// TwinCAT 3 PLC project Untitled1
// ProgramVersion: 3.1.4023.0
// libraries:
//   Tc2_MC2, * (Beckhoff Automation GmbH)
//   Tc2_NC, * (Beckhoff Automation GmbH)
//   Tc2_NCI, * (Beckhoff Automation GmbH)
//   Tc2_PlcInterpolation, * (Beckhoff Automation GmbH)
//   Tc2_Standard, * (Beckhoff Automation GmbH)
//   Tc2_System, * (Beckhoff Automation GmbH)
//   Tc3_Module, * (Beckhoff Automation GmbH)
//   Tc3_mxAutomation, * (Beckhoff Automation GmbH)
//   Tc3_mxAutomationV3_0, * (Beckhoff Automation GmbH)
//   Tc3_mxAutomationV3_1, * (Beckhoff Automation GmbH)
//   Tc3_mxAutomationV3_2, * (Beckhoff Automation GmbH)
//   Tc3_uniValPlc, * (Beckhoff Automation GmbH)
//   Tc3_uniValPlc_v4, * (Beckhoff Automation GmbH)
//   Tc3_uniValPlc_v4_3, * (Beckhoff Automation GmbH)
//   Tc3_uniValPlc_v4_4, * (Beckhoff Automation GmbH)
//   Tc3_uniValPlc_v4_5, * (Beckhoff Automation GmbH)
// project tree:
//   DUTs/ AxisFeedback.TcDUT, AxisInputs.TcDUT
//   GVLs/ Feedback.TcGVL, Inputs.TcGVL, NCI.TcGVL
//   / PlcTask.TcTTO
//   POUs/ AxisControl.TcPOU, FB_EnableAxes.TcPOU, FB_NciFastMFunctions.TcPOU, FB_NciMFunctions.TcPOU, FB_SimpleNciSequence.TcPOU, MAIN.TcPOU, PRG_MFuncControl.TcPOU
// real-time tasks:
//   TASK PlcTask: cycle T#10ms, priority 20, ADS port 350
// motion (NC):
//   TASK NC-Task 1 SAF: cycle T#2ms, priority 4, ADS port 501
//   TASK NC-Task 1 SVB: cycle T#10ms, priority 8, ADS port 511
//   AXIS X (id 1)
//     Dynamic: Acceleration=1505, Deceleration=1505
//     OtherSettings: AllowMotionCmdToSlave=true
//     encoder EncType=1
//     drive DrvType=5
//       TimeComp: TaskDelayCycles=1
//     controller CtrType=1
//       CtrPara: PriorControlFactor=1
//         Observer: BandWidth=20
//   AXIS Y (id 2)
//     OtherSettings: AllowMotionCmdToSlave=true
//     encoder EncType=1
//     drive DrvType=5
//       TimeComp: TaskDelayCycles=1
//     controller CtrType=1
//       CtrPara: PriorControlFactor=1
//         Observer: BandWidth=20
//   AXIS Z (id 3)
//     OtherSettings: AllowMotionCmdToSlave=true
//     encoder EncType=1
//     drive DrvType=5
//       TimeComp: TaskDelayCycles=1
//     controller CtrType=1
//       CtrPara: PriorControlFactor=1
//         Observer: BandWidth=20
//   AXIS Q1 (id 4)
//     Dynamic: VeloJumpFactor=20, ToleranceBallAuxAxis=5
//     OtherSettings: AllowMotionCmdToSlave=true
//     encoder EncType=1
//     drive DrvType=5
//       TimeComp: TaskDelayCycles=1
//     controller CtrType=1
//       CtrPara: PriorControlFactor=1
//         Observer: BandWidth=20
//   AXIS Q2 (id 5)
//     OtherSettings: AllowMotionCmdToSlave=true
//     encoder EncType=1
//     drive DrvType=5
//       TimeComp: TaskDelayCycles=1
//     controller CtrType=1
//       CtrPara: PriorControlFactor=1
//         Observer: BandWidth=20
//   AXIS Q3 (id 6)
//     OtherSettings: AllowMotionCmdToSlave=true
//     encoder EncType=1
//     drive DrvType=5
//       TimeComp: TaskDelayCycles=1
//     controller CtrType=1
//       CtrPara: PriorControlFactor=1
//         Observer: BandWidth=20
// variable links:
//   Untitled1/Untitled1 Instance <-> NC-Task 1 SAF/Axes/Q1
//     PlcTask Inputs/MAIN.io_Q1.NcToPlc <-> Outputs/ToPlc
//     PlcTask Outputs/MAIN.io_Q1.PlcToNc <-> Inputs/FromPlc
//   Untitled1/Untitled1 Instance <-> NC-Task 1 SAF/Axes/Q2
//     PlcTask Inputs/MAIN.io_Q2.NcToPlc <-> Outputs/ToPlc
//     PlcTask Outputs/MAIN.io_Q2.PlcToNc <-> Inputs/FromPlc
//   Untitled1/Untitled1 Instance <-> NC-Task 1 SAF/Axes/Q3
//     PlcTask Inputs/MAIN.io_Q3.NcToPlc <-> Outputs/ToPlc
//     PlcTask Outputs/MAIN.io_Q3.PlcToNc <-> Inputs/FromPlc
//   Untitled1/Untitled1 Instance <-> NC-Task 1 SAF/Axes/X
//     PlcTask Inputs/MAIN.io_X.NcToPlc <-> Outputs/ToPlc
//     PlcTask Outputs/MAIN.io_X.PlcToNc <-> Inputs/FromPlc
//   Untitled1/Untitled1 Instance <-> NC-Task 1 SAF/Axes/Y
//     PlcTask Inputs/MAIN.io_Y.NcToPlc <-> Outputs/ToPlc
//     PlcTask Outputs/MAIN.io_Y.PlcToNc <-> Inputs/FromPlc
//   Untitled1/Untitled1 Instance <-> NC-Task 1 SAF/Axes/Z
//     PlcTask Inputs/MAIN.io_Z.NcToPlc <-> Outputs/ToPlc
//     PlcTask Outputs/MAIN.io_Z.PlcToNc <-> Inputs/FromPlc
//   Untitled1/Untitled1 Instance <-> NC-Task 1 SAF/Interpolation
//     PlcTask Inputs/MAIN.in_stItpToPlc <-> Outputs/ToPlc
//     PlcTask Outputs/MAIN.out_stPlcToItp <-> Inputs/FromPlc

CONFIGURATION Untitled1
    RESOURCE PLC ON TwinCAT3
        TASK PlcTask(INTERVAL := T#10ms, PRIORITY := 20);
        PROGRAM MAIN WITH PlcTask : MAIN;
    END_RESOURCE
END_CONFIGURATION

// ---- DUTs/AxisFeedback.TcDUT
TYPE AxisFeedback :
STRUCT
	Status			: BOOL;
	Busy			: BOOL;
	Active			: BOOL;
	Error			: BOOL;
	ErrorID			: UDINT;	
	Done			: BOOL;
	CommandAborted	: BOOL;
END_STRUCT
END_TYPE

// ---- DUTs/AxisInputs.TcDUT
TYPE AxisInputs :
STRUCT
	PowerEnable		: BOOL;
	EnablePositive	: BOOL;
	EnableNegative  : BOOL;
	Override		: LREAL;
	BufferMode		: MC_BufferMode;
	Options			: ST_PowerOptions;
	
	ResetEnable		: BOOL;
	
	StopExecute			: BOOL;
	StopDeceleration	: LREAL;
	StopJerk			: LREAL;
	StopOptions			: ST_MoveOptions;
	
	
	JogForward		: BOOL;
	JogBackward		: BOOL;
	jogMode			: E_JogMode;
	JogPosition		: LREAL;
	JogVelocity		: LREAL;
	JogAcceleration : LREAL;
	JogDeceleration : LREAL;
	JogJerk			: LREAL;
	
	HaltExecute			: BOOL;
	HaltDeceleration	: LREAL;
	HaltJerk			: LREAL;
	HaltBufferMode		: MC_BufferMode;
	HaltOptions			: ST_MoveOptions;
	
	MoveAbsoluteExecute				: BOOL;
	MoveAbsolutePosition			: LREAL;
	MoveAbsoluteVelocity			: LREAL;
	MoveAbsoluteAcceleration		: LREAL;
	MoveAbsoluteDeceleration		: LREAL;
	MoveAbsoluteJerk				: LREAL;
	MoveAbsoluteBufferMode			: MC_BufferMode;
	MoveAbsoluteOptions				: ST_MoveOptions;
	
	MoveRelativeExecute				: BOOL;
	MoveRelativeDistance			: LREAL;
	MoveRelativeVelocity			: LREAL;
	MoveRelativeAcceleration		: LREAL;
	MoveRelativeDeceleration		: LREAL;
	MoveRelativeJerk				: LREAL;
	MoveRelativeBufferMode			: MC_BufferMode;
	MoveRelativeOptions				: ST_MoveOptions;

END_STRUCT
END_TYPE

// ---- GVLs/Feedback.TcGVL
{attribute 'qualified_only'}
VAR_GLOBAL
	AxisX_Feedback		: AxisFeedback;
	AxisY_Feedback		: AxisFeedback;
	AxisZ_Feedback		: AxisFeedback;
END_VAR

// ---- GVLs/Inputs.TcGVL
{attribute 'qualified_only'}
VAR_GLOBAL
	AxisX_Inputs		: AxisInputs;
	AxisY_Inputs		: AxisInputs;
	AxisZ_Inputs		: AxisInputs;
END_VAR

// ---- GVLs/NCI.TcGVL
{attribute 'qualified_only'}
VAR_GLOBAL
	bMFunc					: ARRAY[0..cnMaxMFuncNumber] OF BOOL;
	bQuitMFunc				: ARRAY[0..cnMaxMFuncNumber] OF BOOL;
	bFastMFunc				: ARRAY[0..cnMaxMFuncNumber] OF BOOL;
END_VAR
VAR_GLOBAL CONSTANT
	cnMaxMFuncNumber		: INT	:= 159;
END_VAR

// ---- POUs/MAIN.TcPOU
PROGRAM MAIN
VAR
	bUserEnableAxes			:	BOOL	:= TRUE;
	fUserOverride			:	LREAL	:= 100.0;
	
	io_X					:	AXIS_REF;
	io_Y					:	AXIS_REF;
	io_Z					:	AXIS_REF;
	io_Q1					:	AXIS_REF;
	io_Q2					:	AXIS_REF;
	io_Q3					:	AXIS_REF;
	
	in_stItpToPlc	AT %I*	:	NcToPlc_NciChannel_Ref;
	out_stPlcToItp	AT %Q*	:	PLCTONC_NCICHANNEL_REF;

	fbEnableAxes			:	FB_EnableAxes;
	bAllAxesReady			:	BOOL;
	
	
	fbSimpleNciSequence		:	FB_SimpleNciSequence;
	bExecSimpleNci			:	BOOL	:= FALSE;
END_VAR

fbEnableAxes(
	bEnableAxes	:= bUserEnableAxes, 
	stX			:=io_X , 
	stY			:=io_Y , 
	stZ			:=io_Z , 
	stM1		:=io_Q1 , 
	stM2		:=io_Q2 , 
	stM3		:=io_Q3 , 
	bAllAxesReady => bAllAxesReady );
	
ItpSetOverridePercent(fOverridePercent:=fUserOverride , sPlcToNci:=out_stPlcToItp);

fbSimpleNciSequence(
	bExecute	:= bExecSimpleNci, 
	bBusy		=> , 
	bError		=> , 
	bDone		=> , 
	stX			:= io_X, 
	stY			:= io_Y, 
	stZ			:= io_Z, 
	stQ1		:= io_Q1,
	stQ2		:= io_Q2,
	stQ3		:= io_Q3,
	stItpToPlc	:= in_stItpToPlc , 
	stPlcToItp	:= out_stPlcToItp);

END_PROGRAM

// ---- POUs/FB_EnableAxes.TcPOU
FUNCTION_BLOCK FB_EnableAxes
VAR_INPUT
	bEnableAxes: BOOL:= TRUE;
END_VAR
VAR_OUTPUT
	bAllAxesReady:	BOOL:= FALSE;
END_VAR
VAR_IN_OUT
	stX:	AXIS_REF;
	stY:	AXIS_REF;
	stZ:	AXIS_REF;
	stM1:	AXIS_REF;
	stM2:	AXIS_REF;
	stM3:	AXIS_REF;
END_VAR
VAR
	fOverride:	LREAL	:= 100.0;
	fbPowerX:	MC_Power;
	fbPowerY:	MC_Power;
	fbPowerZ:	MC_Power;
	fbPowerM1:	MC_Power;
	fbPowerM2:	MC_Power;
	fbPowerM3:	MC_Power;
END_VAR

stX.ReadStatus();
stY.ReadStatus();
stZ.ReadStatus();
stM1.ReadStatus();
stM2.ReadStatus();
stM3.ReadStatus();


fbPowerX(
	Enable:=bEnableAxes, 
	Enable_Positive:=bEnableAxes, 
	Enable_Negative:=bEnableAxes, 
	Override:=fOverride, 
	BufferMode:= , 
	Axis:=stX, 
	Status=> , 
	Busy=> , 
	Active=> , 
	Error=> , 
	ErrorID=> );
fbPowerY(
	Enable:=bEnableAxes, 
	Enable_Positive:=bEnableAxes, 
	Enable_Negative:=bEnableAxes, 
	Override:=fOverride, 
	BufferMode:= , 
	Axis:=stY, 
	Status=> , 
	Busy=> , 
	Active=> , 
	Error=> , 
	ErrorID=> );	
fbPowerZ(
	Enable:=bEnableAxes, 
	Enable_Positive:=bEnableAxes, 
	Enable_Negative:=bEnableAxes, 
	Override:=fOverride, 
	BufferMode:= , 
	Axis:=stZ, 
	Status=> , 
	Busy=> , 
	Active=> , 
	Error=> , 
	ErrorID=> );	
fbPowerM1(
	Enable:=bEnableAxes, 
	Enable_Positive:=bEnableAxes, 
	Enable_Negative:=bEnableAxes, 
	Override:=fOverride, 
	BufferMode:= , 
	Axis:=stM1, 
	Status=> , 
	Busy=> , 
	Active=> , 
	Error=> , 
	ErrorID=> );	
fbPowerM2(
	Enable:=bEnableAxes, 
	Enable_Positive:=bEnableAxes, 
	Enable_Negative:=bEnableAxes, 
	Override:=fOverride, 
	BufferMode:= , 
	Axis:=stM2, 
	Status=> , 
	Busy=> , 
	Active=> , 
	Error=> , 
	ErrorID=> );	
fbPowerM3(
	Enable:=bEnableAxes, 
	Enable_Positive:=bEnableAxes, 
	Enable_Negative:=bEnableAxes, 
	Override:=fOverride, 
	BufferMode:= , 
	Axis:=stM3, 
	Status=> , 
	Busy=> , 
	Active=> , 
	Error=> , 
	ErrorID=> );	
bAllAxesReady	:= fbPowerX.Status AND fbPowerY.Status AND fbPowerZ.Status AND 
	fbPowerM1.Status AND fbPowerM2.Status AND fbPowerM3.Status;

END_FUNCTION_BLOCK

// ---- POUs/FB_SimpleNciSequence.TcPOU
FUNCTION_BLOCK FB_SimpleNciSequence
VAR_INPUT
	bExecute			: BOOL;
END_VAR
VAR_OUTPUT
	bBusy				: BOOL;
	bError				: BOOL;
	bDone				: BOOL;
END_VAR
VAR_IN_OUT
	stX					: AXIS_REF;
	stY					: AXIS_REF;
	stZ					: AXIS_REF;
	stQ1				: AXIS_REF;
	stQ2				: AXIS_REF;
	stQ3				: AXIS_REF;
	stItpToPlc			: NCTOPLC_NCICHANNEL_REF;
	stPlcToItp			: PLCTONC_NCICHANNEL_REF;
END_VAR
VAR
	nState				: UDINT	:= 0;
	nErrorState			: UDINT;
	
	fbBuildGroup		: CfgBuildExt3DGroup;
	fbLoadGCode			: ItpLoadProgEx;
	fbStartGCode		: ItpStartStopEx;
	fbClearGroup		: CfgReconfigGroup;
	fbConfirmHsk		: ItpConfirmHsk;
	
	nInterpreterState	: UDINT	:= 0;
	bConfirmHsk			: BOOL	:= FALSE;
	
//	sPrgName			: STRING(255) := 'GST_SampleFunctions.nc'; //'first.nc';
	sPrgName			: STRING(255) := 'first.nc'; //'';
//	sPrgName			: STRING(255) := 'sample.nc'; //'';
//	sPrgName			: STRING(255) := 'functionsExample.nc'; //'';
	
	
END_VAR

CASE nState OF
0:
	IF bExecute THEN
		bBusy	:= TRUE;
		bDone	:= FALSE;
		bError	:= FALSE;
		nErrorState	:= nState;
		nState	:= 10;
	END_IF	
	
10:
	// first build interpolation group 
	nInterpreterState	:= ItpGetStateInterpreter(sNciToPlc:=stItpToPlc);
	IF nInterpreterState = Tc2_NCI.NCI_INTERPRETER_IDLE THEN
		fbBuildGroup(
			bExecute	:= TRUE, 
			nGroupId	:= ItpGetGroupId(sNciToPlc:=stItpToPlc) , 
			nXAxisId	:= stX.NcToPlc.AxisId, 
			nYAxisId	:= stY.NcToPlc.AxisId, 
			nZAxisId	:= stZ.NcToPlc.AxisId, 
			nQ1AxisId	:= stQ1.NcToPlc.AxisId, 
			nQ2AxisId	:= stQ2.NcToPlc.AxisId, 
			nQ3AxisId	:= stQ3.NcToPlc.AxisId, 
			nQ4AxisId	:= 0, 
			nQ5AxisId	:= 0, 
			tTimeOut	:= , 
			bBusy		=> , 
			bErr		=> , 
			nErrId		=> );
			
		IF NOT fbBuildGroup.bBusy THEN
			IF NOT fbBuildGroup.bErr THEN
				nState	:= 20;
			ELSE
				(* add error handling *)
				nErrorState	:= nState;
				bBusy	:= FALSE;
				bError	:= TRUE;
				nState	:= 9999;
			END_IF
			fbBuildGroup(bExecute:=FALSE); 
		END_IF
	END_IF
	
20:
	// load g-code file 
	// pls. ensure that first.nc is available in TwinCAT\MC\NCI-folder 
	fbLoadGCode(
		sNciToPlc	:= stItpToPlc, 
		bExecute	:= TRUE, 
		sPrg		:= sPrgName, 
		nLength		:= INT_TO_UDINT(LEN(sPrgName)), 
		tTimeOut	:= , 
		bBusy		=> , 
		bErr		=> , 
		nErrId		=> );
		
	IF NOT fbLoadGCode.bBusy THEN
		IF NOT fbLoadGCode.bErr THEN
			nState	:= 30;
		ELSE
			(* add error handling *)
			nErrorState	:= nState;
			bBusy	:= FALSE;
			bError	:= TRUE;
			nState	:= 9999;				
		END_IF
		fbLoadGCode(sNciToPlc:=stItpToPlc, bExecute:=FALSE); 
	END_IF
	
30:
	// we have to check the status of the interpreter. It has to be in ready state, in case of loading the program successfully.
	nInterpreterState	:= ItpGetStateInterpreter(sNciToPlc:=stItpToPlc);
	IF nInterpreterState = Tc2_NCI.NCI_INTERPRETER_READY THEN
		nState	:= 40;
	ELSE
		(* add error handling *)
		nErrorState	:= nState;
		bBusy	:= FALSE;
		bError	:= TRUE;
		nState	:= 9999;				
	END_IF
	
40:
	// start g-code file
	fbStartGCode(
		bStart		:=TRUE, 
		bStop		:=FALSE, 
		tTimeOut	:= , 
		sNciToPlc	:= stItpToPlc, 
		bBusy		=> , 
		bErr		=> , 
		nErrId		=> );
		
	IF NOT fbStartGCode.bBusy THEN
		IF NOT fbStartGCode.bErr THEN
			nState	:= 50;
		ELSE	
			(* add error handling *)
			nErrorState	:= nState;
			bBusy	:= FALSE;
			bError	:= TRUE;
			nState	:= 9999;				
		END_IF
		fbStartGCode( bStart:=FALSE, sNciToPlc:= stItpToPlc ); 
	END_IF
	
50:
	// check state, again - we are at least not in ready state for several ticks
	// this is to ensure that we don't indicate program has finished, before we have started 
	nInterpreterState	:= ItpGetStateInterpreter(sNciToPlc:=stItpToPlc);
	IF nInterpreterState <> Tc2_NCI.NCI_INTERPRETER_READY THEN
		// nci is running
		nState	:= 60;
	END_IF

60:
	nInterpreterState	:= ItpGetStateInterpreter(sNciToPlc:=stItpToPlc);
	IF	nInterpreterState = Tc2_NCI.NCI_INTERPRETER_READY THEN
		// program has finished
		nState	:= 70;
	ELSIF nInterpreterState = Tc2_NCI.NCI_INTERPRETER_ABORTED THEN
		// a run-time error occured - this could be a lag error or something else... 
		// add error handling
		;
	END_IF	
	
70:
	// program has finished 
	// now clear interpolation group 
	fbClearGroup(
		bExecute	:= TRUE, 
		nGroupId	:= ItpGetGroupId(sNciToPlc:=stItpToPlc) , 
		tTimeOut	:= , 
		bBusy		=> , 
		bErr		=> , 
		nErrId		=> );
		
	IF NOT fbClearGroup.bBusy THEN
		IF NOT fbClearGroup.bErr THEN
			nState	:= 80;
		ELSE
			(* add error handling *)
			nErrorState	:= nState;
			bBusy	:= FALSE;
			bError	:= TRUE;
			nState	:= 9999;				
		END_IF
		fbClearGroup(bExecute:=FALSE); 
	END_IF
80:
	bDone	:= TRUE;
	bBusy	:= FALSE;
	IF NOT bExecute THEN
		nState	:= 0;
	END_IF
	
9999:
	// error state 
	IF NOT bExecute THEN
		nState	:= 0;
		bError	:= FALSE;
	END_IF
END_CASE

// handling of m-functions is done outside statemachine
// all m-functions are directly confiremd. In a real application we have of course to consider the m-function numbers to turn on/off certain functions in the machine.
IF ItpIsHskMFunc(stItpToPlc) AND NOT fbConfirmHsk.bBusy THEN
	bConfirmHsk	:= TRUE;
ELSE	
	bConfirmHsk	:= FALSE;
END_IF	

fbConfirmHsk(
	bExecute:=bConfirmHsk , 
	sNciToPlc:=stItpToPlc , 
	sPlcToNci:=stPlcToItp , 
	bBusy=> , 
	bErr=> , 
	nErrId=> );

END_FUNCTION_BLOCK

// ---- POUs/AxisControl.TcPOU
FUNCTION_BLOCK AxisControl
VAR_INPUT
	Axis 			: AXIS_REF;
	AxisInputs		: AxisInputs;
END_VAR
VAR_OUTPUT
	Status			: AxisFeedback;
END_VAR
VAR
	Power			: MC_Power;
	Reset			: MC_Reset;
	Stop			: MC_Stop;
	Jog				: MC_Jog;
	Halt			: MC_Halt;
	MoveAbsolute	: MC_MoveAbsolute;
	MoveRelative	: MC_MoveRelative;
END_VAR

Power(Axis := Axis,
	  Enable := AxisInputs.PowerEnable,
	  Enable_Positive := AxisInputs.EnablePositive,
	  Enable_Negative := AxisInputs.EnableNegative,
	  Override := AxisInputs.Override,
	  BufferMode := AxisInputs.BufferMode,
	  Options := AxisInputs.Options,
	  Status => Status.Status,
	  Busy => Status.Busy,
	  Active => Status.Active,
	  Error => Status.Error,
	  ErrorID => Status.ErrorID);

	 
Reset(Axis := Axis,
	  Execute := AxisInputs.ResetEnable,
	  Done => Status.Done,
      Busy => Status.Busy,
	  Error => Status.Busy,
	  ErrorID => Status.ErrorID);
	  
Stop(Axis := Axis,
	 Execute := AxisInputs.StopExecute,
	 Deceleration := AxisInputs.StopDeceleration,
	 Jerk := AxisInputs.StopJerk,
	 Options := AxisInputs.StopOptions,
	 Done => Status.Done,
	 Busy => Status.Busy,
	 Active => Status.Active,
	 CommandAborted => Status.CommandAborted,
	 Error => Status.Error,
	 ErrorID => Status.ErrorID); 

Halt(Axis := Axis,
	 Execute := AxisInputs.HaltExecute,
	 Deceleration := AxisInputs.HaltDeceleration,
	 Jerk := AxisInputs.HaltJerk,
	 BufferMode := AxisInputs.HaltBufferMode,
	 Options := AxisInputs.HaltOptions,
	 Done => Status.Done,
	 Busy => Status.Busy,
	 Active => Status.Active,
	 CommandAborted => Status.CommandAborted,
	 Error => Status.Error,
	 ErrorID => Status.ErrorID); 

Jog(Axis := Axis,
	JogForward := AxisInputs.JogForward,
	JogBackwards := AxisInputs.JogBackward,
	Mode := AxisInputs.jogMode,
	Position := AxisInputs.JogPosition,
	Velocity := AxisInputs.JogVelocity,
	Acceleration := AxisInputs.JogAcceleration,
	Deceleration := AxisInputs.JogDeceleration,
	jerk := AxisInputs.JogJerk,
	Done => Status.Done,
	Busy => Status.Busy,
	Active => Status.Active,
	CommandAborted => Status.CommandAborted,
	Error => Status.Error,
	ErrorID => Status.ErrorID);
	
MoveAbsolute(Axis := Axis,
			 Execute := AxisInputs.MoveAbsoluteExecute,
			 Position := AxisInputs.MoveAbsolutePosition,
			 Acceleration := AxisInputs.MoveAbsoluteAcceleration,
			 Deceleration := AxisInputs.MoveAbsoluteDeceleration,
			 Jerk := AxisInputs.MoveAbsoluteJerk,
			 Options := AxisInputs.MoveAbsoluteOptions,
			 BufferMode := AxisInputs.MoveAbsoluteBufferMode,
			 Done => Status.Done,
			 Busy => Status.Busy,
			 Active => Status.Active,
			 CommandAborted => Status.CommandAborted,
			 Error => Status.Error,
			 ErrorID => Status.ErrorID);
				 
MoveRelative(Axis := Axis,
			 Execute := AxisInputs.MoveRelativeExecute,
			 Distance := AxisInputs.MoveRelativeDistance,
			 Acceleration := AxisInputs.MoveRelativeAcceleration,
			 Deceleration := AxisInputs.MoveRelativeDeceleration,
			 Jerk := AxisInputs.MoveRelativeJerk,
			 Options := AxisInputs.MoveRelativeOptions,
			 BufferMode := AxisInputs.MoveRelativeBufferMode,
			 Done => Status.Done,
			 Busy => Status.Busy,
			 Active => Status.Active,
			 CommandAborted => Status.CommandAborted,
			 Error => Status.Error,
			 ErrorID => Status.ErrorID);

END_FUNCTION_BLOCK

// ---- POUs/FB_NciFastMFunctions.TcPOU
FUNCTION_BLOCK FB_NciFastMFunctions
VAR_IN_OUT
	sNciToPlc		: NCTOPLC_NCICHANNEL_REF;
END_VAR
VAR_OUTPUT
END_VAR
VAR
	i				: INT;
	l				: SINT;
	bBit			: BOOL;
	index			: UINT;
END_VAR


(* Fill the global defined M-functions array with 
	fast M-Functions from NCI Channel *)

FOR i:=0 TO 4 DO  (* check all 5 dwords *)
	FOR l := 0 TO 31 DO
		bBit := GETBIT32(sNciToPlc.FastMFuncMask[i+1], l);
      	index := INT_TO_UINT((i*32) + l);
		IF ( bBit ) THEN
			NCI.bFastMFunc[index] := TRUE;
		ELSE
			NCI.bFastMFunc[index] := FALSE;
		END_IF
	END_FOR
END_FOR

END_FUNCTION_BLOCK

// ---- POUs/FB_NciMFunctions.TcPOU
FUNCTION_BLOCK FB_NciMFunctions
VAR_IN_OUT
	sNciToPlc		: NCTOPLC_NCICHANNEL_REF;
	sPlcToNci		: PLCTONC_NCICHANNEL_REF;
END_VAR
VAR_OUTPUT
	bBusy			: BOOL;
	bError			: BOOL;
	nErrorId		: UDINT;
END_VAR
VAR
	fbConfirm		: ItpConfirmHsk;
	nAktMfunc		: INT :=  -1;
	bConfirm		: BOOL;
	i				: INT;
END_VAR


(* Check for m function and store information in bMFunc Array	*)
IF ItpIsHskMFunc(sNciToPlc:= sNciToPlc) THEN
	nAktMfunc 			:= ItpGetHskMFunc(sNciToPlc:= sNciToPlc);
	NCI.bMFunc[nAktMfunc]	:= TRUE;
ELSE
	nAktMfunc 	:= -1;
	bConfirm 	:= FALSE;
	FOR i := 0 TO NCI.cnMaxMFuncNumber DO
		NCI.bMFunc[i]		:= FALSE;
		NCI.bQuitMFunc[i]	:= FALSE;
	END_FOR
END_IF

(* Confirm M function, if bit in array bQuitMFunc is set *)
IF nAktMfunc <> -1 THEN
	IF NCI.bQuitMFunc[nAktMfunc] THEN
		bConfirm	:= TRUE;
	END_IF
	NCI.bQuitMFunc[nAktMfunc]	:= FALSE;
END_IF

(* Confirm M function	*)
fbConfirm(
	bExecute	:= bConfirm, 
	sNciToPlc	:= sNciToPlc, 
	sPlcToNci	:= sPlcToNci, 
	bBusy		=> bBusy, 
	bErr		=> bError, 
	nErrId		=> nErrorId);

END_FUNCTION_BLOCK

// ---- POUs/PRG_MFuncControl.TcPOU
PROGRAM PRG_MFuncControl
VAR
	bActivateTool		: BOOL;
END_VAR

IF NCI.bMFunc[5] THEN
	bActivateTool			:= TRUE;
	NCI.bQuitMFunc[11]		:= TRUE;
END_IF


IF NCI.bMFunc[12] THEN
	bActivateTool			:= FALSE;
	NCI.bQuitMFunc[12]		:= TRUE;
END_IF

END_PROGRAM
